// TIA Portal project "RollerConveyorSimulatorIki" (V17)
// Vorlageprojekt für das Buch mit Zielsystem S7-1200

(* hardware
DEVICE "S7-1200-Station_1"  S7-1200 Station
   slot 0: "Baugruppenträger_0"  Rack  V1.0
   slot 1: "PLC_1"  CPU 1211C DC/DC/DC  6ES7 211-1AE40-0XB0  V4.1
*)

// ===== PLC "PLC_1"  CPU 1211C DC/DC/DC =====

VAR_GLOBAL   // PLC tag table "Standard-Variablentabelle"
   "ROLLER CONVEYOR (6M) 1" AT %A0.0 : Bool;
   "STOP" AT %E0.0 : Bool;
   "START" AT %E0.1 : Bool;
   "Tag_4" AT %M0.0 : Bool;
   "Tag_2" AT %M0.1 : Bool;
   "ROLL CONVEYOR (6M) 2" AT %Q0.1 : Bool;
   "DIFFUSE SENSOR 2" AT %I0.2 : Bool;
   "Tag_3" AT %Q0.2 : Bool;
   "Tag_5" AT %Q0.3 : Bool;
   "Tag_6" AT %Q0.4 : Bool;
   "Tag_7" AT %Q0.5 : Bool;
   "DIFFUSE SENSOR 1" AT %I0.3 : Bool;
   "Tag_1" AT %MW2 : Int;
   "Tag_8" AT %M0.2 : Bool;
END_VAR

// folder: System blocks/Program resources

DATA_BLOCK "IEC_Counter_0_DB"   // DB1
{ S7_Optimized_Access := 'TRUE' }
AUTHOR : Simatic
FAMILY : IEC
NAME : CNTR
VERSION : 1.0
// stored: InstanceOfName IEC_COUNTER
"IEC_COUNTER"
BEGIN
END_DATA_BLOCK

DATA_BLOCK "IEC_Timer_0_DB"   // DB2
{ S7_Optimized_Access := 'TRUE' }
AUTHOR : Simatic
FAMILY : IEC
NAME : IEC_TMR
VERSION : 1.0
// stored: InstanceOfName IEC_TIMER
"IEC_TIMER"
BEGIN
END_DATA_BLOCK

// folder: (top level)

FUNCTION "MHJ-PLC-Lab-Function-S71200" : Void   // FC9000, SCL
{ S7_Optimized_Access := 'TRUE' }
VERSION : 0.1
   VAR_TEMP
      rdTimeReturn : Int;
      outputTime : DTL;
      SyncVal : Byte;
      forVal : Int;
      forVal_2 : Int;
      Value : Byte;
   END_VAR
   VAR CONSTANT
      CompVal : Byte := 16#34;
      Value_01 : Byte := 16#11;
      Value_01_DW : DWord := 16#A165_D992;
      Value_02_DW : DWord := 16#58BE_4401;
   END_VAR
BEGIN

   #Value:=PEEK(area := 16#82,
        dbNumber := 0,
        byteOffset := 511);
   #Value := #Value + 1;

   POKE(area := 16#82,
        dbNumber := 0,
        byteOffset := 511,
        value := #Value);

   POKE(area:=16#81,
        dbNumber:=0,
        byteOffset:=1016,
        value:=#Value_01_DW);
   POKE(area := 16#81,
        dbNumber := 0,
        byteOffset := 1020,
        value := #Value_02_DW);

   POKE(area := 16#81,
        dbNumber := 0,
        byteOffset := 511,
        value := B#16#00);

   FOR #forVal := 0 TO 120 DO
       FOR #forVal_2:=0 TO 10 DO
           #rdTimeReturn:=RD_SYS_T(#outputTime);
           #rdTimeReturn := WR_SYS_T(#outputTime);
           #rdTimeReturn := RD_SYS_T(#outputTime);
           #rdTimeReturn := WR_SYS_T(#outputTime);
       END_FOR;
       #SyncVal:= PEEK(area := 16#81,
                      dbNumber := 0,
                      byteOffset := 511);
       IF #SyncVal = #CompVal THEN
          GOTO M_1;
       END_IF;
   END_FOR;
   RETURN;

   M_1:
   POKE(area := 16#81,
        dbNumber := 0,
        byteOffset := 511,
        value := B#16#0);
END_FUNCTION

ORGANIZATION_BLOCK "Main"   // OB1, LAD, ProgramCycle
TITLE = "Main Program Sweep (Cycle)"
{ S7_Optimized_Access := 'TRUE' }
VERSION : 0.1
   VAR_INPUT
      Initial_Call : Bool;   // Initial call of this OB
      Remanence : Bool;   // =True, if remanent data are available
   END_VAR
BEGIN

REGION Network 1: Konnektierungsbaustein für PLC-Lab
   // Im Netzwerk 1 wird der Konnektierungsbaustein für PLC-Lab aufgerufen.
   // Dieser Aufruf darf nicht entfernt werden!
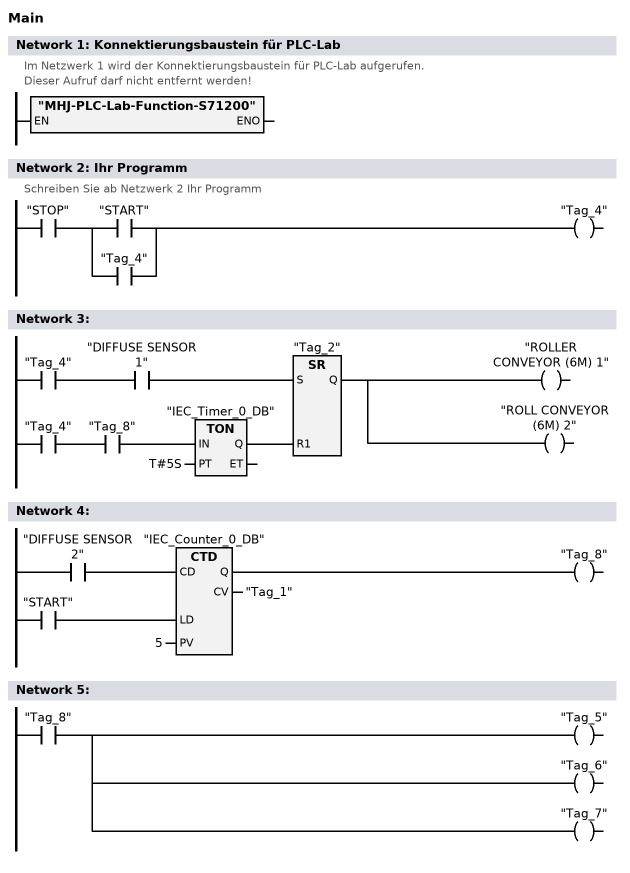
   RUNG wire#powerrail
      "MHJ-PLC-Lab-Function-S71200"()
   END_RUNG
   // the same network as SCL:
   "MHJ-PLC-Lab-Function-S71200"();
END_REGION

REGION Network 2: Ihr Programm
   // Schreiben Sie ab Netzwerk 2 Ihr Programm
   RUNG wire#powerrail
      Contact( "STOP" )
      wire#w1
      Contact( "START" )
      wire#w2
      Coil( "Tag_4" )
   END_RUNG
   RUNG wire#w1
      Contact( "Tag_4" )
   END_RUNG wire#w2
   // the same network as SCL:
   "Tag_4" := "STOP" AND ("START" OR "Tag_4");
END_REGION

REGION Network 3
   "IEC_Timer_0_DB".TON(IN := "Tag_4" AND "Tag_8", PT := T#5S);
   IF "Tag_4" AND "DIFFUSE SENSOR 1" THEN
       "Tag_2" := TRUE;   // SR flip-flop
   END_IF;
   IF "IEC_Timer_0_DB".Q THEN "Tag_2" := FALSE; END_IF;
   "ROLLER CONVEYOR (6M) 1" := "Tag_2";
   "ROLL CONVEYOR (6M) 2" := "Tag_2";
END_REGION

REGION Network 4
   "IEC_Counter_0_DB".CTD(CD := "DIFFUSE SENSOR 2", LD := "START", PV := 5, CV => "Tag_1");
   "Tag_8" := "IEC_Counter_0_DB".Q;
END_REGION

REGION Network 5
   RUNG wire#powerrail
      Contact( "Tag_8" )
      wire#w1
      Coil( "Tag_5" )
   END_RUNG
   RUNG wire#w1
      Coil( "Tag_6" )
   END_RUNG
   RUNG wire#w1
      Coil( "Tag_7" )
   END_RUNG
   // the same network as SCL:
   "Tag_5" := "Tag_8";
   "Tag_6" := "Tag_8";
   "Tag_7" := "Tag_8";
END_REGION
END_ORGANIZATION_BLOCK